// TIA Portal project "Llenadora de botellas" (V15)

(* hardware
DEVICE "S71500/ET200MP station_1"  S7-1500 station
   slot 0: "Perfil soporte_0"  Rack  6ES7 590-1***0-0AA0
   slot 1: "PLC_1"  CPU 1512C-1 PN  6ES7 512-1CK01-0AB0  V2.5
      slot 3: "Display de la CPU_1"  6ES7591-1AA00-0AA0
*)

// ===== PLC "PLC_1"  CPU 1512C-1 PN =====

VAR_GLOBAL   // PLC tag table "Motor"
   "TimerAlarma" AT %T1 : Timer;   // Sirve como temporizador para las alarmas de FB motor
END_VAR

TYPE "Secuencia"
   STRUCT
      Start : Bool;
      Stop : Bool;
      Etapa : Int;
      EtapaAnterior : Int;
      Temporizadores_TONR : Array[1..16] of TONR_TIME;
      SalidasTemporizadores : Array[1..16] of Bool;
      Flancos : Array[1..16] of Bool;
   END_STRUCT;
END_TYPE

// folder: 01_Entradas/Salidas

DATA_BLOCK "Entradas"   // DB2
{ S7_Optimized_Access := 'TRUE' }
VERSION : 0.1
   VAR
      Disyuntor : Bool;
      Start : Bool;
      Stop : Bool;
      Sensor1 : Bool;
      Sensor2 : Bool;
   END_VAR
BEGIN
END_DATA_BLOCK

DATA_BLOCK "Salidas"   // DB3
{ S7_Optimized_Access := 'TRUE' }
VERSION : 0.1
   VAR
      Motores : Array[1..8] of Bool;
   END_VAR
BEGIN
END_DATA_BLOCK

// folder: 02_Linea de embotellado

DATA_BLOCK "MotorBanda"   // DB1
{ S7_Optimized_Access := 'TRUE' }
VERSION : 0.1
// stored: InstanceOfName FB_Motor
"FB_Motor"
BEGIN
END_DATA_BLOCK

DATA_BLOCK "Tramos"   // DB100
{ S7_Optimized_Access := 'TRUE' }
VERSION : 0.1
   VAR
      Tramo : Array[1..16] of "Secuencia";
      ConteoBotellas : Array[1..16] of Int;
   END_VAR
BEGIN
END_DATA_BLOCK

// folder: (top level)

ORGANIZATION_BLOCK "Main"   // OB1, LAD, ProgramCycle
TITLE = "Main Program Sweep (Cycle)"
{ S7_Optimized_Access := 'TRUE' }
VERSION : 0.1
   VAR_INPUT
      Initial_Call : Bool;   // Initial call of this OB
      Remanence : Bool;   // =True, if remanent data are available
   END_VAR
BEGIN

REGION Network 1
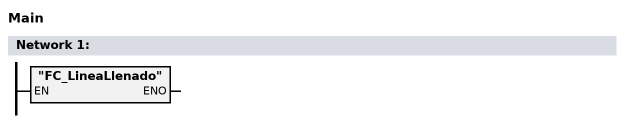
   RUNG wire#powerrail
      "FC_LineaLlenado"()
   END_RUNG
   // the same network as SCL:
   "FC_LineaLlenado"();
END_REGION
END_ORGANIZATION_BLOCK

// folder: 00_Bloques estándar/FB

FUNCTION_BLOCK "FB_Motor"   // FB1, LAD
TITLE = -----------------------------------|> NOTA INICIAL
{ S7_Optimized_Access := 'TRUE' }
VERSION : 0.1
// Cualquier cambio a la FB en sus variables debe ser precedido por tomar una instántanea del o los DB de instancia individual si esta en funcionamiento. Ya que de lo contrario esto puede llevar a un mal funcionamiento del sistema.
   VAR_INPUT
      StartManual : Bool;   // Entrada de arranque por botón en panel de control
      StartAutomatic : Bool;   // Entrada de arranque por HMI
      Disyuntor : Bool;
   END_VAR
   VAR_OUTPUT
      MarchaMotor : Bool;
   END_VAR
   VAR
      HMI : Struct   // Valores que maneja la HMI
         Start : Bool;   // Arranque del motor desde pantalla
         segTrabajo : Int;
         minTrabajo : Int;
         HorTrabajo : Int;
      END_STRUCT;
      Habilitador : Bool;
      Alarma : Array[1..16] of Bool;
      Rearme : Bool;
      "Timer" : Array[1..16] of TON_TIME;
      Timer_ET : Array[1..16] of Time;
      Timer_ON : Array[1..16] of Bool;
      PermisoExterno : Bool;
   END_VAR
   VAR_TEMP
      EnMarcha : Bool;
      EstadoAlarmas : Bool;
   END_VAR
   VAR_TEMP   // added for the SCL form of the ladder/FBD networks
      _w1 : Bool;
      _w2 : Bool;
   END_VAR
BEGIN

REGION Network 1 (STL): -----------------------------------| Habilitación del motor |-----------------------------------
         A     #StartManual;
         O(;
         A     #StartAutomatic;
         A     #HMI.Start;
         );
         =     #Habilitador;
END_REGION

NETWORK
TITLE = -----------------------------------| Alarmas de seguridad |-----------------------------------

REGION Network 3 (STL): -----------------------------------|> Alarma 1 - Breaker (disyuntor)
   // Si el motor esta habilitado entonces se activa la alarma pero para evitar un posible mal funcionamiento del contactor se coloca un temporizador de 1 segundo para evitar que la alarma se este encendiendo y apagando bruscamente.
         A     #Habilitador;  // Contacto abierto del habilitador del motor
         A     #Disyuntor;
         L     S5T#1S;  // Cargamos tiempo de 1 segundo
         SF    "TimerAlarma";  // Configura el temporizador
         A     "TimerAlarma";  // Guarda el valor de salida del temporizador

         O(;
         A     #Alarma[1];
         AN    #Rearme;
         );
         =     #Alarma[1];  // Habilita la alarma
END_REGION

REGION Network 4: -----------------------------------|> Alarma 2 - Vacía
END_REGION

REGION Network 5: -----------------------------------|> Alarma 3 - Vacía
END_REGION

REGION Network 6 (SCL): -----------------------------------| Marcha del motor |-----------------------------------
END_REGION

REGION Network 7 (STL): -----------------------------------|> Verificación de alarmas
         AN    #Alarma[1];
         AN    #Alarma[2];
         AN    #Alarma[3];
         AN    #Alarma[4];
         AN    #Alarma[5];
         AN    #Alarma[6];
         AN    #Alarma[7];
         AN    #Alarma[8];
         AN    #Alarma[9];
         AN    #Alarma[10];
         AN    #Alarma[11];
         AN    #Alarma[12];
         AN    #Alarma[13];
         AN    #Alarma[14];
         AN    #Alarma[15];
         AN    #Alarma[16];
         =     #EstadoAlarmas;  // 0 -> Alguna alarma activada y 1 -> Sin alarmas
END_REGION

REGION Network 8: -----------------------------------|> Puesta en marcha del motor
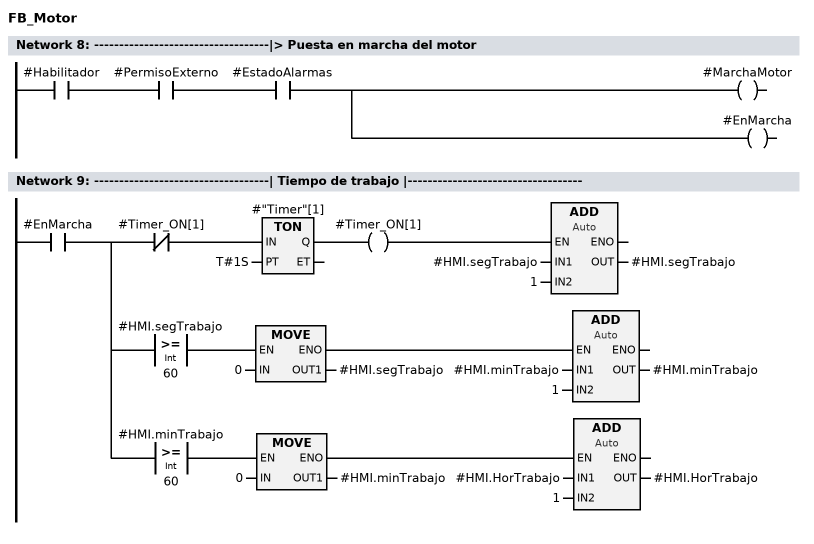
   RUNG wire#powerrail
      Contact( #Habilitador )
      Contact( #PermisoExterno )
      Contact( #EstadoAlarmas )
      wire#w1
      Coil( #MarchaMotor )
   END_RUNG
   RUNG wire#w1
      Coil( #EnMarcha )
   END_RUNG
   // the same network as SCL:
   #MarchaMotor := #Habilitador AND #PermisoExterno AND #EstadoAlarmas;
   #EnMarcha := #MarchaMotor;
END_REGION

REGION Network 9: -----------------------------------| Tiempo de trabajo |-----------------------------------
   #"Timer"[1].TON(IN := #EnMarcha AND NOT #Timer_ON[1], PT := T#1S);
   #Timer_ON[1] := #"Timer"[1].Q;
   IF #"Timer"[1].Q THEN #HMI.segTrabajo := #HMI.segTrabajo + 1; END_IF;
   #_w1 := #EnMarcha AND (#HMI.segTrabajo >= 60);
   IF #_w1 THEN
       #HMI.segTrabajo := 0;
       #HMI.minTrabajo := #HMI.minTrabajo + 1;
   END_IF;
   #_w2 := #EnMarcha AND (#HMI.minTrabajo >= 60);
   IF #_w2 THEN
       #HMI.minTrabajo := 0;
       #HMI.HorTrabajo := #HMI.HorTrabajo + 1;
   END_IF;
END_REGION
END_FUNCTION_BLOCK

// folder: 02_Linea de embotellado

FUNCTION "FC_LineaLlenado" : Void   // FC100, LAD
{ S7_Optimized_Access := 'TRUE' }
VERSION : 0.1
BEGIN

REGION Network 1: -----------------------------------| Linea de llenado |-----------------------------------
END_REGION

REGION Network 2 (STL)

   // Se llaman las funciones que ponen en marcha a los tramos

         CALL  "FC_Tramo1_Llenado"
         ( PermisoMotor := "MotorBanda".PermisoExterno,
           T1           := "Tramos".Tramo[1]
         );



         CALL  "FC_Tramo2_Llenado"
         ( T2 := "Tramos".Tramo[2]
         );


   // Se llama al FB motor cuya instancia individual es MotorBanda [DB1]

   //-----------------------------------------
   // StartManual    -> Iniciar por medio de botón
   // StartAutomatic -> Inicia desde una HMI
   //------------------------------------------

         CALL  "FB_Motor", "MotorBanda"
         ( StartManual    := FALSE,
           StartAutomatic := TRUE,
           Disyuntor      := "Entradas".Disyuntor,
           MarchaMotor    := "Salidas".Motores[1]
         );
END_REGION
END_FUNCTION

// folder: Tramo1

FUNCTION "FC_Tramo1_Llenado" : Void   // FC101, LAD
{ S7_Optimized_Access := 'TRUE' }
VERSION : 0.1
// LA ETAPA INICIAL 0, ETAPA 2, ETAPA 3 Y STOP DETIENEN AL MOTOR
   VAR_OUTPUT
      PermisoMotor : Bool;
   END_VAR
   VAR_IN_OUT
      T1 : "Secuencia";
   END_VAR
   VAR CONSTANT
      EtapaStopSeguridad : Int := 911;
   END_VAR
   VAR_TEMP   // added for the SCL form of the ladder/FBD networks
      _w1 : Bool;
   END_VAR
BEGIN

REGION Network 1: -----------------------------------| Funcionamiento del primer tramo |-----------------------------------
END_REGION

REGION Network 2: -----------------------------------|> Etapa inicial (0 -----> 1)
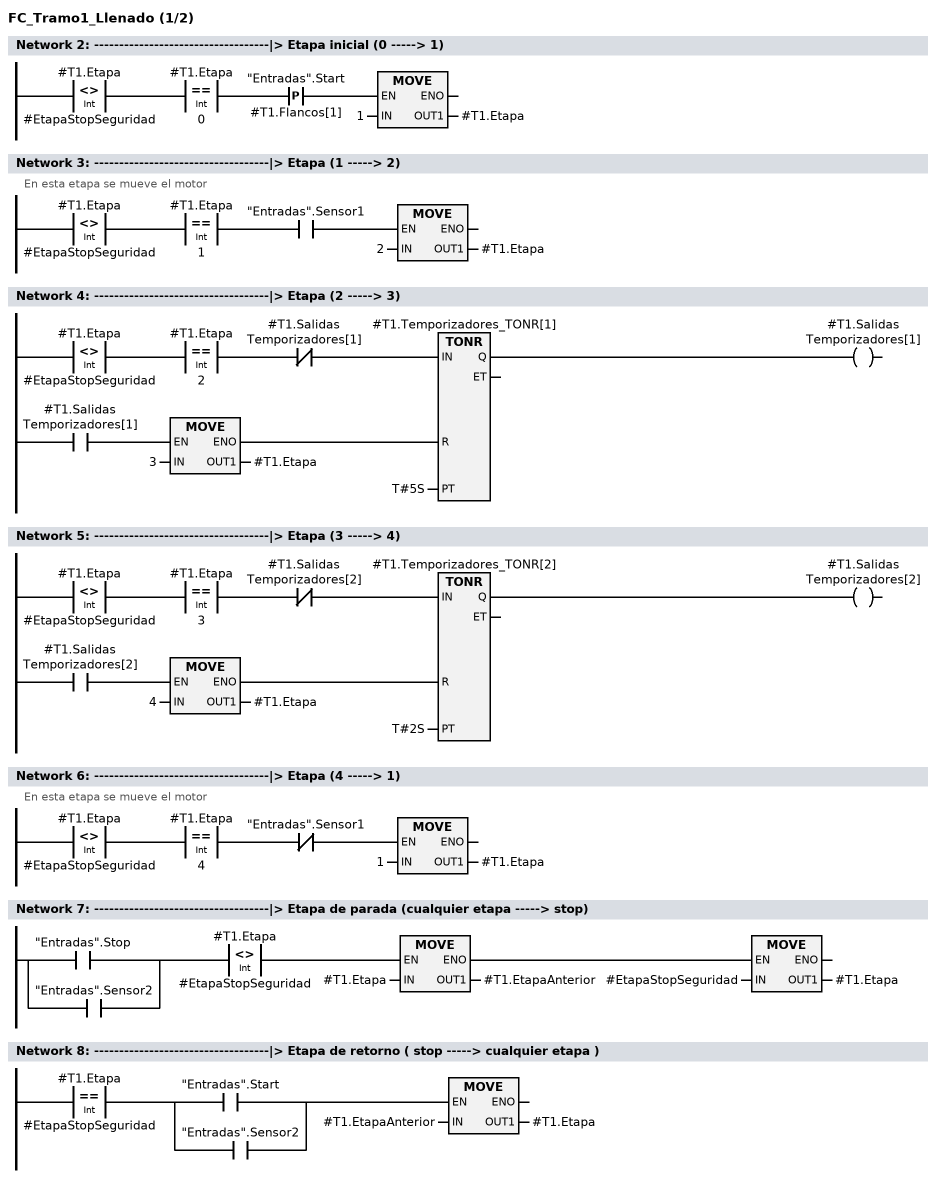
   RUNG wire#powerrail
      { S7_Templates := "SrcType := Int" } NE_Contact(in1 := #T1.Etapa, in2 := #EtapaStopSeguridad)
      { S7_Templates := "SrcType := Int" } EQ_Contact(in1 := #T1.Etapa, in2 := 0)
      P_Contact(operand := "Entradas".Start, bit := #T1.Flancos[1])
      Move(in := 1, out1 => #T1.Etapa)
   END_RUNG
   // the same network as SCL:
   #_w1 := (#T1.Etapa <> #EtapaStopSeguridad) AND (#T1.Etapa = 0) AND "Entradas".Start AND NOT #T1.Flancos[1];   // rising edge of "Entradas".Start
   #T1.Flancos[1] := "Entradas".Start;
   IF #_w1 THEN #T1.Etapa := 1; END_IF;
END_REGION

REGION Network 3: -----------------------------------|> Etapa (1 -----> 2)
   // En esta etapa se mueve el motor
   RUNG wire#powerrail
      { S7_Templates := "SrcType := Int" } NE_Contact(in1 := #T1.Etapa, in2 := #EtapaStopSeguridad)
      { S7_Templates := "SrcType := Int" } EQ_Contact(in1 := #T1.Etapa, in2 := 1)
      Contact( "Entradas".Sensor1 )
      Move(in := 2, out1 => #T1.Etapa)
   END_RUNG
   // the same network as SCL:
   IF (#T1.Etapa <> #EtapaStopSeguridad) AND (#T1.Etapa = 1) AND "Entradas".Sensor1 THEN
       #T1.Etapa := 2;
   END_IF;
END_REGION

REGION Network 4: -----------------------------------|> Etapa (2 -----> 3)
   #_w1 := (#T1.Etapa <> #EtapaStopSeguridad) AND (#T1.Etapa = 2) AND NOT #T1.SalidasTemporizadores[1];
   IF #T1.SalidasTemporizadores[1] THEN #T1.Etapa := 3; END_IF;
   #T1.Temporizadores_TONR[1].TONR(IN := #_w1, R := #T1.SalidasTemporizadores[1], PT := T#5S);
   #T1.SalidasTemporizadores[1] := #T1.Temporizadores_TONR[1].Q;
END_REGION

REGION Network 5: -----------------------------------|> Etapa (3 -----> 4)
   #_w1 := (#T1.Etapa <> #EtapaStopSeguridad) AND (#T1.Etapa = 3) AND NOT #T1.SalidasTemporizadores[2];
   IF #T1.SalidasTemporizadores[2] THEN #T1.Etapa := 4; END_IF;
   #T1.Temporizadores_TONR[2].TONR(IN := #_w1, R := #T1.SalidasTemporizadores[2], PT := T#2S);
   #T1.SalidasTemporizadores[2] := #T1.Temporizadores_TONR[2].Q;
END_REGION

REGION Network 6: -----------------------------------|> Etapa (4 -----> 1)
   // En esta etapa se mueve el motor
   RUNG wire#powerrail
      { S7_Templates := "SrcType := Int" } NE_Contact(in1 := #T1.Etapa, in2 := #EtapaStopSeguridad)
      { S7_Templates := "SrcType := Int" } EQ_Contact(in1 := #T1.Etapa, in2 := 4)
      I_Contact( "Entradas".Sensor1 )
      Move(in := 1, out1 => #T1.Etapa)
   END_RUNG
   // the same network as SCL:
   IF (#T1.Etapa <> #EtapaStopSeguridad) AND (#T1.Etapa = 4) AND NOT "Entradas".Sensor1 THEN
       #T1.Etapa := 1;
   END_IF;
END_REGION

REGION Network 7: -----------------------------------|> Etapa de parada (cualquier etapa -----> stop)
   RUNG wire#powerrail
      Contact( "Entradas".Stop )
      wire#w1
      { S7_Templates := "SrcType := Int" } NE_Contact(in1 := #T1.Etapa, in2 := #EtapaStopSeguridad)
      Move(in := #T1.Etapa, out1 => #T1.EtapaAnterior)
      Move(in := #EtapaStopSeguridad, out1 => #T1.Etapa)
   END_RUNG
   RUNG wire#powerrail
      Contact( "Entradas".Sensor2 )
   END_RUNG wire#w1
   // the same network as SCL:
   IF ("Entradas".Stop OR "Entradas".Sensor2) AND (#T1.Etapa <> #EtapaStopSeguridad) THEN
       #T1.EtapaAnterior := #T1.Etapa;
       #T1.Etapa := #EtapaStopSeguridad;
   END_IF;
END_REGION

REGION Network 8: -----------------------------------|> Etapa de retorno ( stop -----> cualquier etapa )
   RUNG wire#powerrail
      { S7_Templates := "SrcType := Int" } EQ_Contact(in1 := #T1.Etapa, in2 := #EtapaStopSeguridad)
      wire#w1
      Contact( "Entradas".Start )
      wire#w2
      Move(in := #T1.EtapaAnterior, out1 => #T1.Etapa)
   END_RUNG
   RUNG wire#w1
      Contact( "Entradas".Sensor2 )
   END_RUNG wire#w2
   // the same network as SCL:
   IF (#T1.Etapa = #EtapaStopSeguridad) AND ("Entradas".Start OR "Entradas".Sensor2) THEN
       #T1.Etapa := #T1.EtapaAnterior;
   END_IF;
END_REGION

REGION Network 9: -----------------------------------|> Conteo de botellas igual a 10 regresa el proceso a la etapa inicial
   // Hay que ponerle un retardo por si llega al final para que termine de llenar de azucar en el tramo 2 (creo)
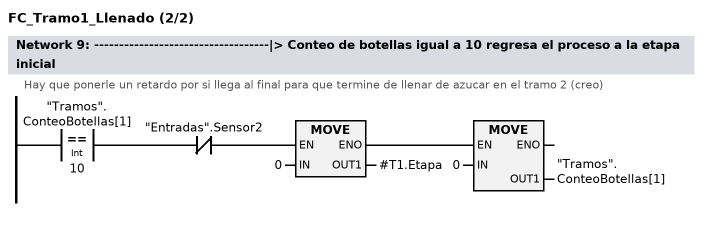
   RUNG wire#powerrail
      { S7_Templates := "SrcType := Int" } EQ_Contact(in1 := "Tramos".ConteoBotellas[1], in2 := 10)
      I_Contact( "Entradas".Sensor2 )
      Move(in := 0, out1 => #T1.Etapa)
      Move(in := 0, out1 => "Tramos".ConteoBotellas[1])
   END_RUNG
   // the same network as SCL:
   IF ("Tramos".ConteoBotellas[1] = 10) AND NOT "Entradas".Sensor2 THEN
       #T1.Etapa := 0;
       "Tramos".ConteoBotellas[1] := 0;
   END_IF;
END_REGION

REGION Network 10 (STL): -----------------------------------|> Permiso de marcha para el motor
   // Si se encuentra en la etapa 1 o en la etapa 4 se pone en marcha el motor

         A(;
         L     #T1.Etapa;
         L     1;
         ==I;
         );
         O(;
         L     #T1.Etapa;
         L     4;
         ==I;
         );
         =     #PermisoMotor;
END_REGION
END_FUNCTION

// folder: Tramo2

FUNCTION "FC_Tramo2_Llenado" : Void   // FC102, LAD
{ S7_Optimized_Access := 'TRUE' }
VERSION : 0.1
   VAR_IN_OUT
      T2 : "Secuencia";
   END_VAR
   VAR CONSTANT
      EtapaStopSeguridad : Int := 911;
   END_VAR
   VAR_TEMP   // added for the SCL form of the ladder/FBD networks
      _w1 : Bool;
   END_VAR
BEGIN

REGION Network 1: -----------------------------------| Funcionamiento del segundo tramo |-----------------------------------
END_REGION

REGION Network 2: -----------------------------------|> Etapa inicial (0 -----> 1)
   // En esta etapa funciona el motor
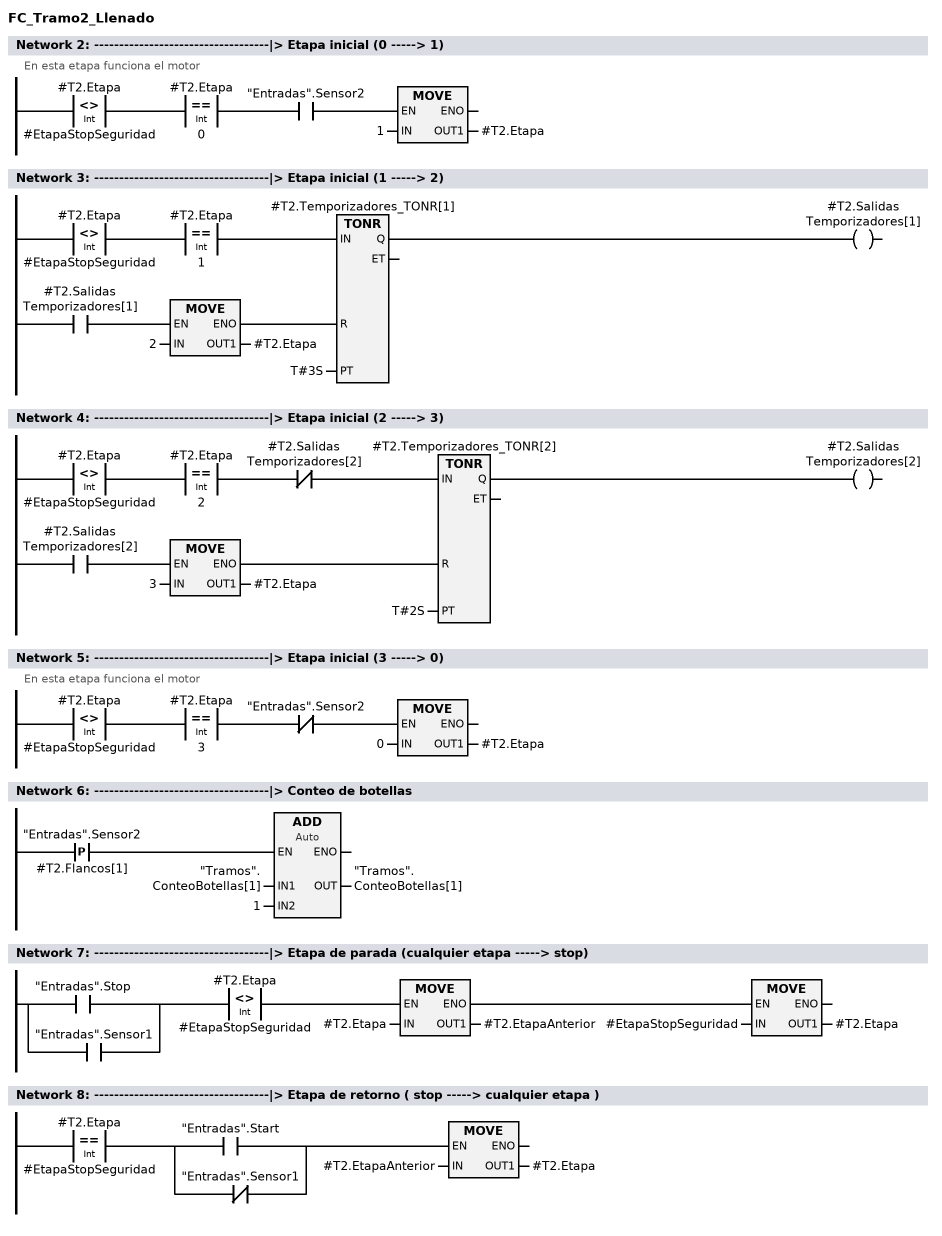
   RUNG wire#powerrail
      { S7_Templates := "SrcType := Int" } NE_Contact(in1 := #T2.Etapa, in2 := #EtapaStopSeguridad)
      { S7_Templates := "SrcType := Int" } EQ_Contact(in1 := #T2.Etapa, in2 := 0)
      Contact( "Entradas".Sensor2 )
      Move(in := 1, out1 => #T2.Etapa)
   END_RUNG
   // the same network as SCL:
   IF (#T2.Etapa <> #EtapaStopSeguridad) AND (#T2.Etapa = 0) AND "Entradas".Sensor2 THEN
       #T2.Etapa := 1;
   END_IF;
END_REGION

REGION Network 3: -----------------------------------|> Etapa inicial (1 -----> 2)
   #_w1 := (#T2.Etapa <> #EtapaStopSeguridad) AND (#T2.Etapa = 1);
   IF #T2.SalidasTemporizadores[1] THEN #T2.Etapa := 2; END_IF;
   #T2.Temporizadores_TONR[1].TONR(IN := #_w1, R := #T2.SalidasTemporizadores[1], PT := T#3S);
   #T2.SalidasTemporizadores[1] := #T2.Temporizadores_TONR[1].Q;
END_REGION

REGION Network 4: -----------------------------------|> Etapa inicial (2 -----> 3)
   #_w1 := (#T2.Etapa <> #EtapaStopSeguridad) AND (#T2.Etapa = 2) AND NOT #T2.SalidasTemporizadores[2];
   IF #T2.SalidasTemporizadores[2] THEN #T2.Etapa := 3; END_IF;
   #T2.Temporizadores_TONR[2].TONR(IN := #_w1, R := #T2.SalidasTemporizadores[2], PT := T#2S);
   #T2.SalidasTemporizadores[2] := #T2.Temporizadores_TONR[2].Q;
END_REGION

REGION Network 5: -----------------------------------|> Etapa inicial (3 -----> 0)
   // En esta etapa funciona el motor
   RUNG wire#powerrail
      { S7_Templates := "SrcType := Int" } NE_Contact(in1 := #T2.Etapa, in2 := #EtapaStopSeguridad)
      { S7_Templates := "SrcType := Int" } EQ_Contact(in1 := #T2.Etapa, in2 := 3)
      I_Contact( "Entradas".Sensor2 )
      Move(in := 0, out1 => #T2.Etapa)
   END_RUNG
   // the same network as SCL:
   IF (#T2.Etapa <> #EtapaStopSeguridad) AND (#T2.Etapa = 3) AND NOT "Entradas".Sensor2 THEN
       #T2.Etapa := 0;
   END_IF;
END_REGION

REGION Network 6: -----------------------------------|> Conteo de botellas
   RUNG wire#powerrail
      P_Contact(operand := "Entradas".Sensor2, bit := #T2.Flancos[1])
      Add(in1 := "Tramos".ConteoBotellas[1], in2 := 1, out => "Tramos".ConteoBotellas[1])
   END_RUNG
   // the same network as SCL:
   #_w1 := "Entradas".Sensor2 AND NOT #T2.Flancos[1];   // rising edge of "Entradas".Sensor2
   #T2.Flancos[1] := "Entradas".Sensor2;
   IF #_w1 THEN "Tramos".ConteoBotellas[1] := "Tramos".ConteoBotellas[1] + 1; END_IF;
END_REGION

REGION Network 7: -----------------------------------|> Etapa de parada (cualquier etapa -----> stop)
   RUNG wire#powerrail
      Contact( "Entradas".Stop )
      wire#w1
      { S7_Templates := "SrcType := Int" } NE_Contact(in1 := #T2.Etapa, in2 := #EtapaStopSeguridad)
      Move(in := #T2.Etapa, out1 => #T2.EtapaAnterior)
      Move(in := #EtapaStopSeguridad, out1 => #T2.Etapa)
   END_RUNG
   RUNG wire#powerrail
      Contact( "Entradas".Sensor1 )
   END_RUNG wire#w1
   // the same network as SCL:
   IF ("Entradas".Stop OR "Entradas".Sensor1) AND (#T2.Etapa <> #EtapaStopSeguridad) THEN
       #T2.EtapaAnterior := #T2.Etapa;
       #T2.Etapa := #EtapaStopSeguridad;
   END_IF;
END_REGION

REGION Network 8: -----------------------------------|> Etapa de retorno ( stop -----> cualquier etapa )
   RUNG wire#powerrail
      { S7_Templates := "SrcType := Int" } EQ_Contact(in1 := #T2.Etapa, in2 := #EtapaStopSeguridad)
      wire#w1
      Contact( "Entradas".Start )
      wire#w2
      Move(in := #T2.EtapaAnterior, out1 => #T2.Etapa)
   END_RUNG
   RUNG wire#w1
      I_Contact( "Entradas".Sensor1 )
   END_RUNG wire#w2
   // the same network as SCL:
   IF (#T2.Etapa = #EtapaStopSeguridad) AND ("Entradas".Start OR NOT "Entradas".Sensor1) THEN
       #T2.Etapa := #T2.EtapaAnterior;
   END_IF;
END_REGION

REGION Network 9 (STL): -----------------------------------|> Permiso de marcha para el motor
   // Si se pone en la etapa 0 o en la 3 se pone en marcha el motor

   //U(
   //L     #T2.Etapa
   //L     0
   //==I
   //)
   //O(
   //L     #T2.Etapa
   //L     3
   //==I
   //)
   //=     #PermisoMotor        // Este permiso se puede omitir
END_REGION
END_FUNCTION